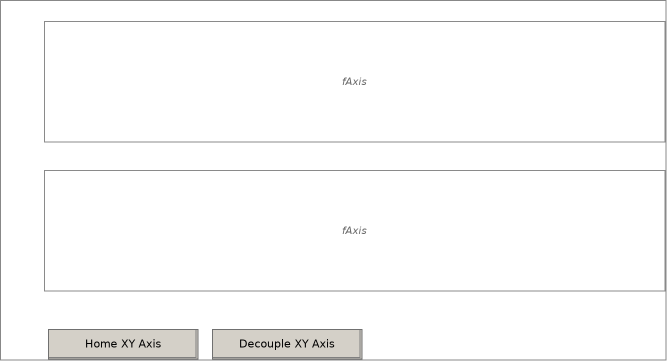
VISUALIZATION Visualization  // 667x361
    Frame (44,21 621x121)
        shows fAxis(io_fbAxis := MAIN.fbXAxis)
    Frame (44,170 621x121)
        shows fAxis(io_fbAxis := MAIN.fbYAxis)
    Button (48,329 150x30), "Home XY Axis"
        toggle MAIN.bHomeXYAxis
    Button (212,329 150x30), "Decouple XY Axis"
        toggle MAIN.bDecoupleXYAxis
END_VISUALIZATION

(* stored: Version 1.1.0.1, ProductVersion 3.1.4024.2
   Visu Visualization: Id {c808b8ff-45ec-41a6-942a-efd22e83f903} *)
